(* Schneider Machine Expert - Basic project Questao3.4_FelipeV1_20241009, file version 2.9.0.0 *)
(* ProjectInformations: Name=Novo projeto *)

HARDWARE
  Cpu 0: TM221M16R/G
  ModuleExtensionObject 0: TM3DM24R/G
  EthernetConfiguration: NetworkName=M221, IpAllocationMode=FixedAddress, IpAddress=0.0.0.0, SubnetMask=0.0.0.0
  SerialLineConfiguration: Baud=Baud19200, Parity=ParityEven, DataBits=DataBits8, StopBits=StopBits1, PhysicalMedium=PhysicalMediumRs485, TransmissionMode=TransmissionModeModbusRtu, SlaveId=1, Addressing=SlaveAddressing
  MastTask: UsePeriodScanMode=false, PeriodScan=100
  FastTask: Period=255
  CpuBehavior: StartingMode=StartAsPreviousState, AutoSaveRamOnEeprom=true, WatchdogPeriod=250

SYMBOLS  (address, symbol, comment, settings)
  %M0       L_ATUA
  %M1       L_DESA
  %M2       D_ATUA
  %M3       D_DESA
  %M4       INIC_SENSOR_A
  %M5       INIC_SENSOR_B
  %M6       INIC_SENSOR_C
  %M7       INIC_CHAV_SEL_P
  %M8       INIC_CHAV_SEL_M
  %M9       INIC_CHAV_SEL_G
  %M15      SENSOR_ERRO
  %M20      ESTEIRA_LIGA
  %M21      ESTEIRA_DESL
  %M22      ALAR_AL_LIGA
  %M23      ALAR_AL_DESL
  %I0.0     BOT_L_ATUA
  %I0.1     BOT_L_DESA
  %I0.2     BOT_D_ATUA
  %I0.3     BOT_D_DESA
  %I0.4     SENSOR_A
  %I0.5     SENSOR_B
  %I0.6     SENSOR_C
  %I0.7     CHAV_SELEC_P
  %Q0.1     ESTEIRA
  %Q0.2     ALARME_AL
  %I1.0     CHAV_SELEC_M
  %I1.1     CHAV_SELEC_G

POU Novo POU
  (* SectionNumber=0 *)

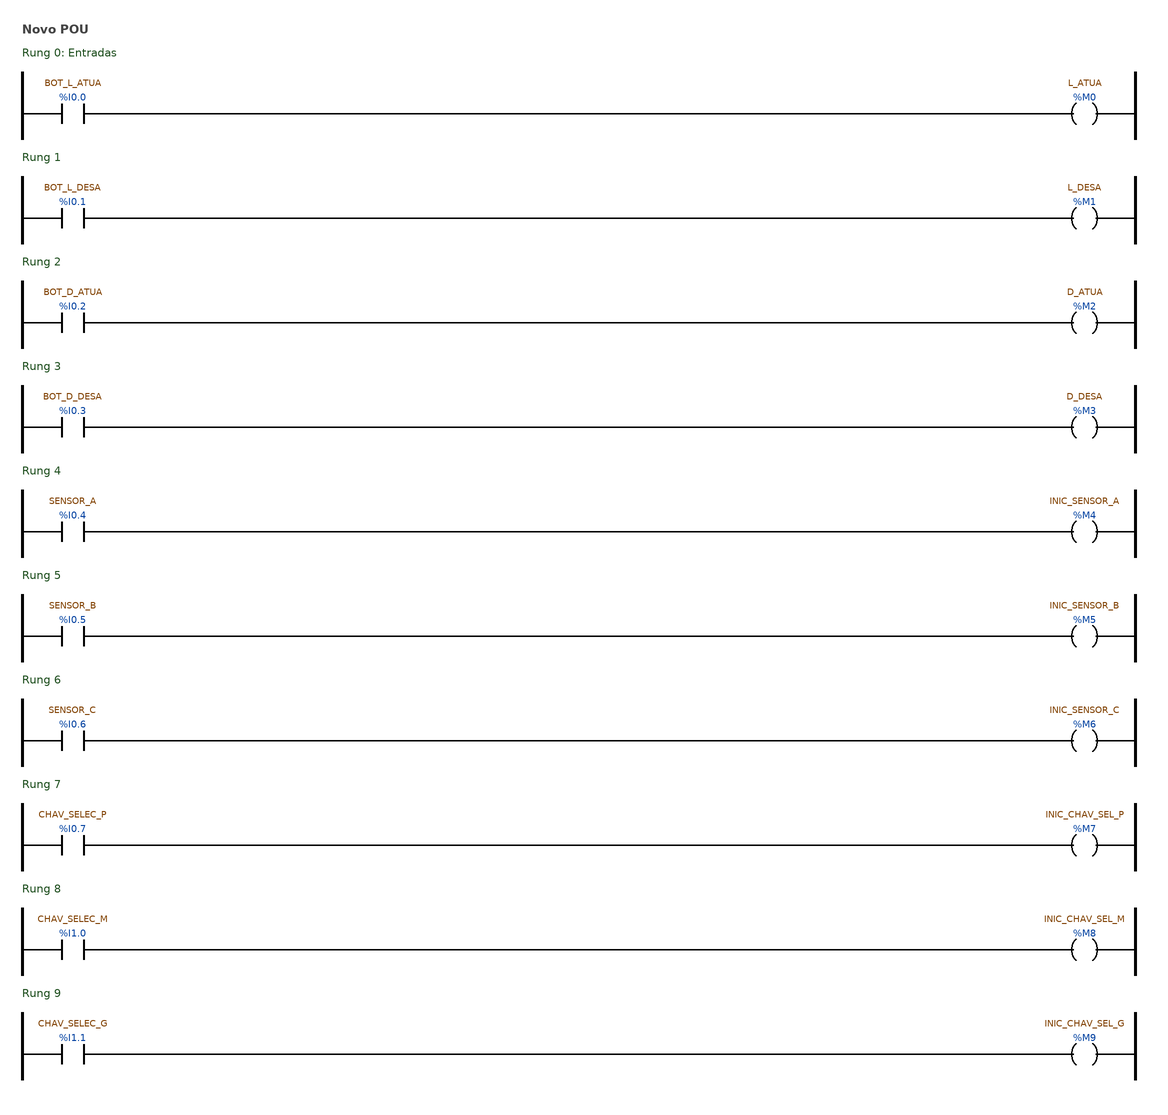

// Rung 0: Entradas
  LD %I0.0                (* BOT_L_ATUA *)
  ST %M0                  (* L_ATUA *)
  // as ST:
  //   L_ATUA := BOT_L_ATUA;

// Rung 1
  LD %I0.1                (* BOT_L_DESA *)
  ST %M1                  (* L_DESA *)
  // as ST:
  //   L_DESA := BOT_L_DESA;

// Rung 2
  LD %I0.2                (* BOT_D_ATUA *)
  ST %M2                  (* D_ATUA *)
  // as ST:
  //   D_ATUA := BOT_D_ATUA;

// Rung 3
  LD %I0.3                (* BOT_D_DESA *)
  ST %M3                  (* D_DESA *)
  // as ST:
  //   D_DESA := BOT_D_DESA;

// Rung 4
  LD %I0.4                (* SENSOR_A *)
  ST %M4                  (* INIC_SENSOR_A *)
  // as ST:
  //   INIC_SENSOR_A := SENSOR_A;

// Rung 5
  LD %I0.5                (* SENSOR_B *)
  ST %M5                  (* INIC_SENSOR_B *)
  // as ST:
  //   INIC_SENSOR_B := SENSOR_B;

// Rung 6
  LD %I0.6                (* SENSOR_C *)
  ST %M6                  (* INIC_SENSOR_C *)
  // as ST:
  //   INIC_SENSOR_C := SENSOR_C;

// Rung 7
  LD %I0.7                (* CHAV_SELEC_P *)
  ST %M7                  (* INIC_CHAV_SEL_P *)
  // as ST:
  //   INIC_CHAV_SEL_P := CHAV_SELEC_P;

// Rung 8
  LD %I1.0                (* CHAV_SELEC_M *)
  ST %M8                  (* INIC_CHAV_SEL_M *)
  // as ST:
  //   INIC_CHAV_SEL_M := CHAV_SELEC_M;

// Rung 9
  LD %I1.1                (* CHAV_SELEC_G *)
  ST %M9                  (* INIC_CHAV_SEL_G *)
  // as ST:
  //   INIC_CHAV_SEL_G := CHAV_SELEC_G;

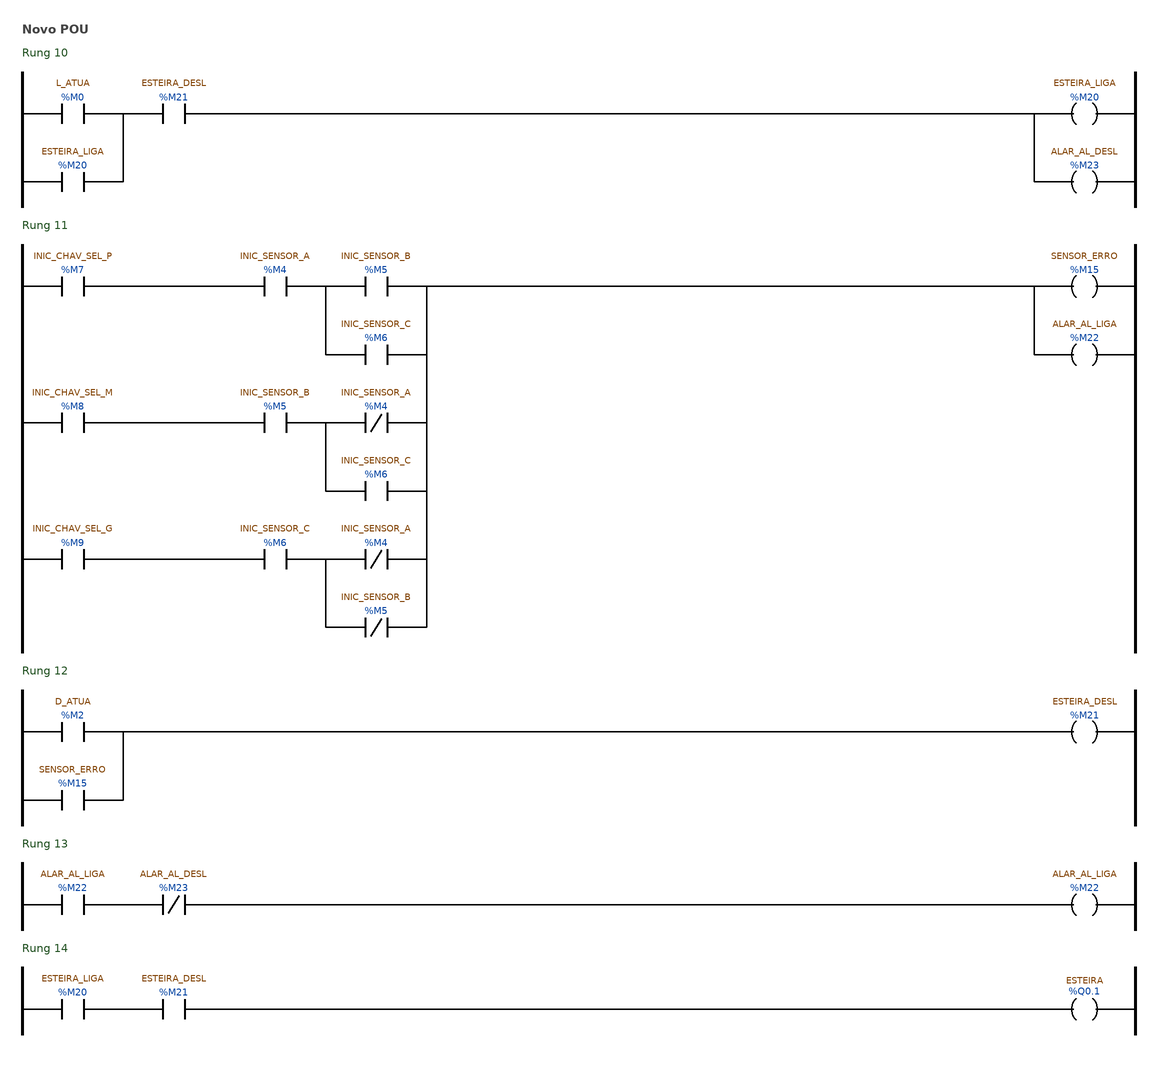

// Rung 10
  LD %M0                  (* L_ATUA *)
  OR %M20                 (* ESTEIRA_LIGA *)
  AND %M21                (* ESTEIRA_DESL *)
  ST %M20                 (* ESTEIRA_LIGA *)
  ST %M23                 (* ALAR_AL_DESL *)
  // as ST:
  //   _t1 := (L_ATUA OR ESTEIRA_LIGA) AND ESTEIRA_DESL;
  //   ESTEIRA_LIGA := _t1;
  //   ALAR_AL_DESL := _t1;

// Rung 11
  LD %M7                  (* INIC_CHAV_SEL_P *)
  AND %M4                 (* INIC_SENSOR_A *)
  AND( %M5                (* INIC_SENSOR_B *)
  OR %M6                  (* INIC_SENSOR_C *)
  )
  OR( %M8                 (* INIC_CHAV_SEL_M *)
  AND %M5                 (* INIC_SENSOR_B *)
  AND(N %M4               (* INIC_SENSOR_A *)
  OR %M6                  (* INIC_SENSOR_C *)
  )
  )
  OR( %M9                 (* INIC_CHAV_SEL_G *)
  AND %M6                 (* INIC_SENSOR_C *)
  AND(N %M4               (* INIC_SENSOR_A *)
  ORN %M5                 (* INIC_SENSOR_B *)
  )
  )
  ST %M15                 (* SENSOR_ERRO *)
  ST %M22                 (* ALAR_AL_LIGA *)
  // as ST:
  //   SENSOR_ERRO := INIC_CHAV_SEL_P AND INIC_SENSOR_A AND (INIC_SENSOR_B OR INIC_SENSOR_C) OR INIC_CHAV_SEL_M AND INIC_SENSOR_B AND (NOT INIC_SENSOR_A OR INIC_SENSOR_C) OR INIC_CHAV_SEL_G AND INIC_SENSOR_C AND (NOT INIC_SENSOR_A OR NOT INIC_SENSOR_B);
  //   ALAR_AL_LIGA := INIC_CHAV_SEL_P AND INIC_SENSOR_A AND (INIC_SENSOR_B OR INIC_SENSOR_C) OR INIC_CHAV_SEL_M AND INIC_SENSOR_B AND (NOT INIC_SENSOR_A OR INIC_SENSOR_C) OR INIC_CHAV_SEL_G AND INIC_SENSOR_C AND (NOT INIC_SENSOR_A OR NOT INIC_SENSOR_B);

// Rung 12
  LD %M2                  (* D_ATUA *)
  OR %M15                 (* SENSOR_ERRO *)
  ST %M21                 (* ESTEIRA_DESL *)
  // as ST:
  //   ESTEIRA_DESL := D_ATUA OR SENSOR_ERRO;

// Rung 13
  LD %M22                 (* ALAR_AL_LIGA *)
  ANDN %M23               (* ALAR_AL_DESL *)
  ST %M22                 (* ALAR_AL_LIGA *)
  // as ST:
  //   ALAR_AL_LIGA := ALAR_AL_LIGA AND NOT ALAR_AL_DESL;

// Rung 14
  LD %M20                 (* ESTEIRA_LIGA *)
  AND %M21                (* ESTEIRA_DESL *)
  ST %Q0.1                (* ESTEIRA *)
  // as ST:
  //   ESTEIRA := ESTEIRA_LIGA AND ESTEIRA_DESL;

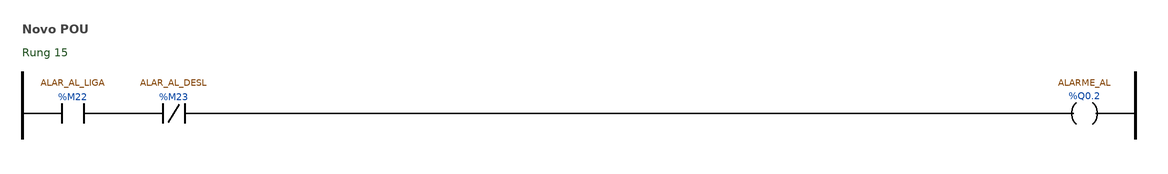

// Rung 15
  LD %M22                 (* ALAR_AL_LIGA *)
  ANDN %M23               (* ALAR_AL_DESL *)
  ST %Q0.2                (* ALARME_AL *)
  // as ST:
  //   ALARME_AL := ALAR_AL_LIGA AND NOT ALAR_AL_DESL;
